// TIA Portal V18 export
// export: Created 2026-06-13T06:09:36.1107387Z, ExportSetting WithDefaults, DisplayName Totally Integrated Automation Portal, DisplayVersion V18, DisplayName TIA Portal Openness, DisplayVersion V18, DisplayName TIA Portal Version Control Interface, DisplayVersion V18, DisplayName STEP 7 Professional, DisplayVersion V18, DisplayName STEP 7 Safety, DisplayVersion V18, DisplayName WinCC Professional, DisplayVersion V18
FUNCTION "FC_HMI_Mirror_PLC2" : Void   // FC41, LAD
{ S7_Optimized_Access := 'TRUE' }
VERSION : 0.1
// stored: AutoNumber true, IsIECCheckEnabled false, SetENOAutomatically false, UDAEnableTagReadback false
BEGIN

REGION Network 1: Mirror AI_V3240_Nuoc_Bon3
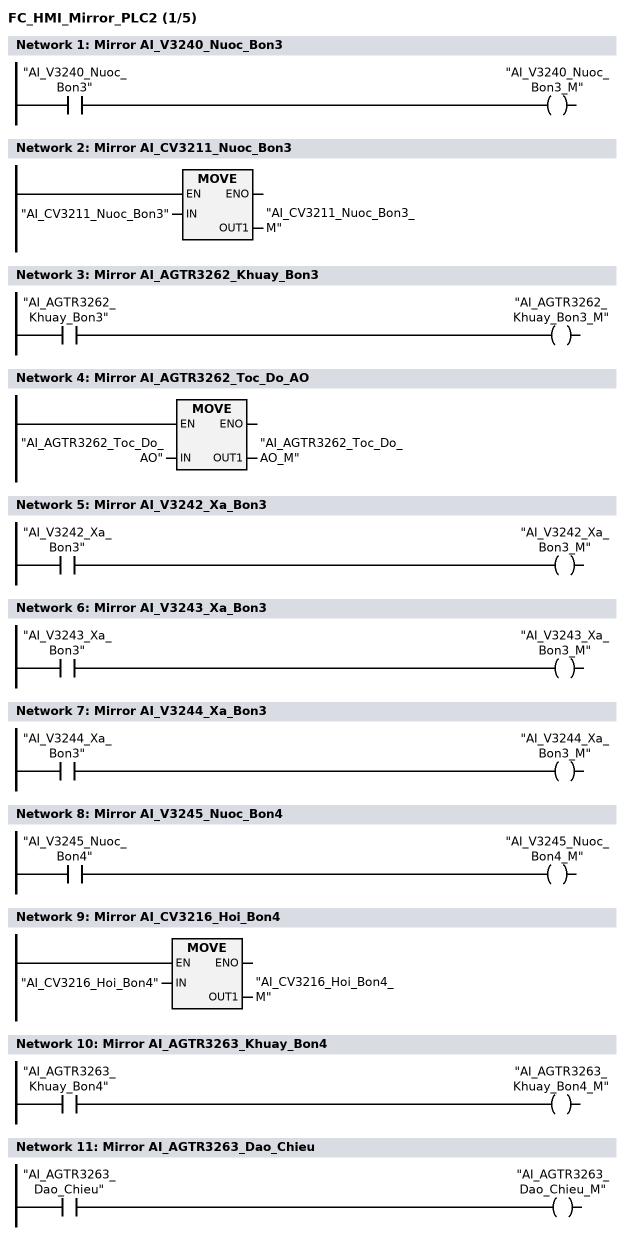
   RUNG wire#powerrail
      Contact( "AI_V3240_Nuoc_Bon3" )
      Coil( "AI_V3240_Nuoc_Bon3_M" )
   END_RUNG
   // the same network as SCL:
   "AI_V3240_Nuoc_Bon3_M" := "AI_V3240_Nuoc_Bon3";
END_REGION

REGION Network 2: Mirror AI_CV3211_Nuoc_Bon3
   RUNG wire#powerrail
      { S7_GenerateENO := "TRUE" } Move(in := "AI_CV3211_Nuoc_Bon3", out1 => "AI_CV3211_Nuoc_Bon3_M")
   END_RUNG
   // the same network as SCL:
   "AI_CV3211_Nuoc_Bon3_M" := "AI_CV3211_Nuoc_Bon3";
END_REGION

REGION Network 3: Mirror AI_AGTR3262_Khuay_Bon3
   RUNG wire#powerrail
      Contact( "AI_AGTR3262_Khuay_Bon3" )
      Coil( "AI_AGTR3262_Khuay_Bon3_M" )
   END_RUNG
   // the same network as SCL:
   "AI_AGTR3262_Khuay_Bon3_M" := "AI_AGTR3262_Khuay_Bon3";
END_REGION

REGION Network 4: Mirror AI_AGTR3262_Toc_Do_AO
   RUNG wire#powerrail
      { S7_GenerateENO := "TRUE" } Move(in := "AI_AGTR3262_Toc_Do_AO", out1 => "AI_AGTR3262_Toc_Do_AO_M")
   END_RUNG
   // the same network as SCL:
   "AI_AGTR3262_Toc_Do_AO_M" := "AI_AGTR3262_Toc_Do_AO";
END_REGION

REGION Network 5: Mirror AI_V3242_Xa_Bon3
   RUNG wire#powerrail
      Contact( "AI_V3242_Xa_Bon3" )
      Coil( "AI_V3242_Xa_Bon3_M" )
   END_RUNG
   // the same network as SCL:
   "AI_V3242_Xa_Bon3_M" := "AI_V3242_Xa_Bon3";
END_REGION

REGION Network 6: Mirror AI_V3243_Xa_Bon3
   RUNG wire#powerrail
      Contact( "AI_V3243_Xa_Bon3" )
      Coil( "AI_V3243_Xa_Bon3_M" )
   END_RUNG
   // the same network as SCL:
   "AI_V3243_Xa_Bon3_M" := "AI_V3243_Xa_Bon3";
END_REGION

REGION Network 7: Mirror AI_V3244_Xa_Bon3
   RUNG wire#powerrail
      Contact( "AI_V3244_Xa_Bon3" )
      Coil( "AI_V3244_Xa_Bon3_M" )
   END_RUNG
   // the same network as SCL:
   "AI_V3244_Xa_Bon3_M" := "AI_V3244_Xa_Bon3";
END_REGION

REGION Network 8: Mirror AI_V3245_Nuoc_Bon4
   RUNG wire#powerrail
      Contact( "AI_V3245_Nuoc_Bon4" )
      Coil( "AI_V3245_Nuoc_Bon4_M" )
   END_RUNG
   // the same network as SCL:
   "AI_V3245_Nuoc_Bon4_M" := "AI_V3245_Nuoc_Bon4";
END_REGION

REGION Network 9: Mirror AI_CV3216_Hoi_Bon4
   RUNG wire#powerrail
      { S7_GenerateENO := "TRUE" } Move(in := "AI_CV3216_Hoi_Bon4", out1 => "AI_CV3216_Hoi_Bon4_M")
   END_RUNG
   // the same network as SCL:
   "AI_CV3216_Hoi_Bon4_M" := "AI_CV3216_Hoi_Bon4";
END_REGION

REGION Network 10: Mirror AI_AGTR3263_Khuay_Bon4
   RUNG wire#powerrail
      Contact( "AI_AGTR3263_Khuay_Bon4" )
      Coil( "AI_AGTR3263_Khuay_Bon4_M" )
   END_RUNG
   // the same network as SCL:
   "AI_AGTR3263_Khuay_Bon4_M" := "AI_AGTR3263_Khuay_Bon4";
END_REGION

REGION Network 11: Mirror AI_AGTR3263_Dao_Chieu
   RUNG wire#powerrail
      Contact( "AI_AGTR3263_Dao_Chieu" )
      Coil( "AI_AGTR3263_Dao_Chieu_M" )
   END_RUNG
   // the same network as SCL:
   "AI_AGTR3263_Dao_Chieu_M" := "AI_AGTR3263_Dao_Chieu";
END_REGION

REGION Network 12: Mirror AI_AGTR3263_Toc_Do_AO
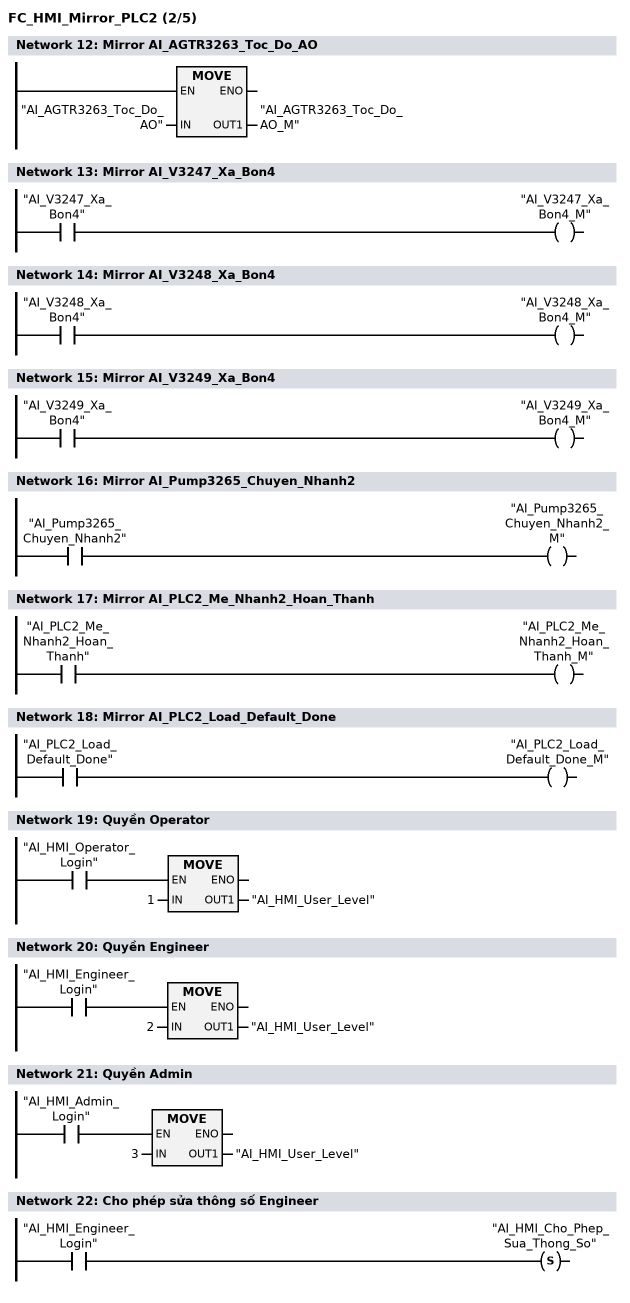
   RUNG wire#powerrail
      { S7_GenerateENO := "TRUE" } Move(in := "AI_AGTR3263_Toc_Do_AO", out1 => "AI_AGTR3263_Toc_Do_AO_M")
   END_RUNG
   // the same network as SCL:
   "AI_AGTR3263_Toc_Do_AO_M" := "AI_AGTR3263_Toc_Do_AO";
END_REGION

REGION Network 13: Mirror AI_V3247_Xa_Bon4
   RUNG wire#powerrail
      Contact( "AI_V3247_Xa_Bon4" )
      Coil( "AI_V3247_Xa_Bon4_M" )
   END_RUNG
   // the same network as SCL:
   "AI_V3247_Xa_Bon4_M" := "AI_V3247_Xa_Bon4";
END_REGION

REGION Network 14: Mirror AI_V3248_Xa_Bon4
   RUNG wire#powerrail
      Contact( "AI_V3248_Xa_Bon4" )
      Coil( "AI_V3248_Xa_Bon4_M" )
   END_RUNG
   // the same network as SCL:
   "AI_V3248_Xa_Bon4_M" := "AI_V3248_Xa_Bon4";
END_REGION

REGION Network 15: Mirror AI_V3249_Xa_Bon4
   RUNG wire#powerrail
      Contact( "AI_V3249_Xa_Bon4" )
      Coil( "AI_V3249_Xa_Bon4_M" )
   END_RUNG
   // the same network as SCL:
   "AI_V3249_Xa_Bon4_M" := "AI_V3249_Xa_Bon4";
END_REGION

REGION Network 16: Mirror AI_Pump3265_Chuyen_Nhanh2
   RUNG wire#powerrail
      Contact( "AI_Pump3265_Chuyen_Nhanh2" )
      Coil( "AI_Pump3265_Chuyen_Nhanh2_M" )
   END_RUNG
   // the same network as SCL:
   "AI_Pump3265_Chuyen_Nhanh2_M" := "AI_Pump3265_Chuyen_Nhanh2";
END_REGION

REGION Network 17: Mirror AI_PLC2_Me_Nhanh2_Hoan_Thanh
   RUNG wire#powerrail
      Contact( "AI_PLC2_Me_Nhanh2_Hoan_Thanh" )
      Coil( "AI_PLC2_Me_Nhanh2_Hoan_Thanh_M" )
   END_RUNG
   // the same network as SCL:
   "AI_PLC2_Me_Nhanh2_Hoan_Thanh_M" := "AI_PLC2_Me_Nhanh2_Hoan_Thanh";
END_REGION

REGION Network 18: Mirror AI_PLC2_Load_Default_Done
   RUNG wire#powerrail
      Contact( "AI_PLC2_Load_Default_Done" )
      Coil( "AI_PLC2_Load_Default_Done_M" )
   END_RUNG
   // the same network as SCL:
   "AI_PLC2_Load_Default_Done_M" := "AI_PLC2_Load_Default_Done";
END_REGION

REGION Network 19: Quyền Operator
   RUNG wire#powerrail
      Contact( "AI_HMI_Operator_Login" )
      { S7_GenerateENO := "TRUE" } Move(in := 1, out1 => "AI_HMI_User_Level")
   END_RUNG
   // the same network as SCL:
   IF "AI_HMI_Operator_Login" THEN "AI_HMI_User_Level" := 1; END_IF;
END_REGION

REGION Network 20: Quyền Engineer
   RUNG wire#powerrail
      Contact( "AI_HMI_Engineer_Login" )
      { S7_GenerateENO := "TRUE" } Move(in := 2, out1 => "AI_HMI_User_Level")
   END_RUNG
   // the same network as SCL:
   IF "AI_HMI_Engineer_Login" THEN "AI_HMI_User_Level" := 2; END_IF;
END_REGION

REGION Network 21: Quyền Admin
   RUNG wire#powerrail
      Contact( "AI_HMI_Admin_Login" )
      { S7_GenerateENO := "TRUE" } Move(in := 3, out1 => "AI_HMI_User_Level")
   END_RUNG
   // the same network as SCL:
   IF "AI_HMI_Admin_Login" THEN "AI_HMI_User_Level" := 3; END_IF;
END_REGION

REGION Network 22: Cho phép sửa thông số Engineer
   RUNG wire#powerrail
      Contact( "AI_HMI_Engineer_Login" )
      S_Coil( "AI_HMI_Cho_Phep_Sua_Thong_So" )
   END_RUNG
   // the same network as SCL:
   IF "AI_HMI_Engineer_Login" THEN "AI_HMI_Cho_Phep_Sua_Thong_So" := TRUE; END_IF;
END_REGION

REGION Network 23: Cho phép sửa thông số Admin
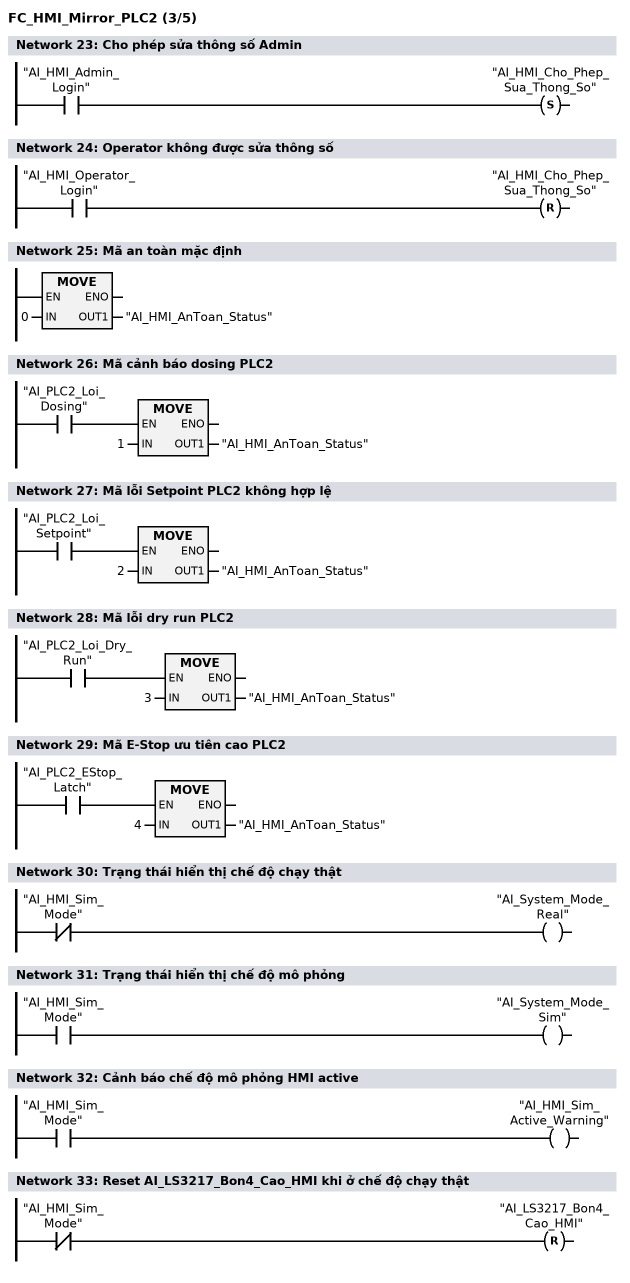
   RUNG wire#powerrail
      Contact( "AI_HMI_Admin_Login" )
      S_Coil( "AI_HMI_Cho_Phep_Sua_Thong_So" )
   END_RUNG
   // the same network as SCL:
   IF "AI_HMI_Admin_Login" THEN "AI_HMI_Cho_Phep_Sua_Thong_So" := TRUE; END_IF;
END_REGION

REGION Network 24: Operator không được sửa thông số
   RUNG wire#powerrail
      Contact( "AI_HMI_Operator_Login" )
      R_Coil( "AI_HMI_Cho_Phep_Sua_Thong_So" )
   END_RUNG
   // the same network as SCL:
   IF "AI_HMI_Operator_Login" THEN "AI_HMI_Cho_Phep_Sua_Thong_So" := FALSE; END_IF;
END_REGION

REGION Network 25: Mã an toàn mặc định
   RUNG wire#powerrail
      { S7_GenerateENO := "TRUE" } Move(in := 0, out1 => "AI_HMI_AnToan_Status")
   END_RUNG
   // the same network as SCL:
   "AI_HMI_AnToan_Status" := 0;
END_REGION

REGION Network 26: Mã cảnh báo dosing PLC2
   RUNG wire#powerrail
      Contact( "AI_PLC2_Loi_Dosing" )
      { S7_GenerateENO := "TRUE" } Move(in := 1, out1 => "AI_HMI_AnToan_Status")
   END_RUNG
   // the same network as SCL:
   IF "AI_PLC2_Loi_Dosing" THEN "AI_HMI_AnToan_Status" := 1; END_IF;
END_REGION

REGION Network 27: Mã lỗi Setpoint PLC2 không hợp lệ
   RUNG wire#powerrail
      Contact( "AI_PLC2_Loi_Setpoint" )
      { S7_GenerateENO := "TRUE" } Move(in := 2, out1 => "AI_HMI_AnToan_Status")
   END_RUNG
   // the same network as SCL:
   IF "AI_PLC2_Loi_Setpoint" THEN "AI_HMI_AnToan_Status" := 2; END_IF;
END_REGION

REGION Network 28: Mã lỗi dry run PLC2
   RUNG wire#powerrail
      Contact( "AI_PLC2_Loi_Dry_Run" )
      { S7_GenerateENO := "TRUE" } Move(in := 3, out1 => "AI_HMI_AnToan_Status")
   END_RUNG
   // the same network as SCL:
   IF "AI_PLC2_Loi_Dry_Run" THEN "AI_HMI_AnToan_Status" := 3; END_IF;
END_REGION

REGION Network 29: Mã E-Stop ưu tiên cao PLC2
   RUNG wire#powerrail
      Contact( "AI_PLC2_EStop_Latch" )
      { S7_GenerateENO := "TRUE" } Move(in := 4, out1 => "AI_HMI_AnToan_Status")
   END_RUNG
   // the same network as SCL:
   IF "AI_PLC2_EStop_Latch" THEN "AI_HMI_AnToan_Status" := 4; END_IF;
END_REGION

REGION Network 30: Trạng thái hiển thị chế độ chạy thật
   RUNG wire#powerrail
      I_Contact( "AI_HMI_Sim_Mode" )
      Coil( "AI_System_Mode_Real" )
   END_RUNG
   // the same network as SCL:
   "AI_System_Mode_Real" := NOT "AI_HMI_Sim_Mode";
END_REGION

REGION Network 31: Trạng thái hiển thị chế độ mô phỏng
   RUNG wire#powerrail
      Contact( "AI_HMI_Sim_Mode" )
      Coil( "AI_System_Mode_Sim" )
   END_RUNG
   // the same network as SCL:
   "AI_System_Mode_Sim" := "AI_HMI_Sim_Mode";
END_REGION

REGION Network 32: Cảnh báo chế độ mô phỏng HMI active
   RUNG wire#powerrail
      Contact( "AI_HMI_Sim_Mode" )
      Coil( "AI_HMI_Sim_Active_Warning" )
   END_RUNG
   // the same network as SCL:
   "AI_HMI_Sim_Active_Warning" := "AI_HMI_Sim_Mode";
END_REGION

REGION Network 33: Reset AI_LS3217_Bon4_Cao_HMI khi ở chế độ chạy thật
   RUNG wire#powerrail
      I_Contact( "AI_HMI_Sim_Mode" )
      R_Coil( "AI_LS3217_Bon4_Cao_HMI" )
   END_RUNG
   // the same network as SCL:
   IF NOT "AI_HMI_Sim_Mode" THEN "AI_LS3217_Bon4_Cao_HMI" := FALSE; END_IF;
END_REGION

REGION Network 34: Reset AI_Pump3265_Chuyen_Nhanh2_Cmd_Nhan_HMI khi ở chế độ chạy thật
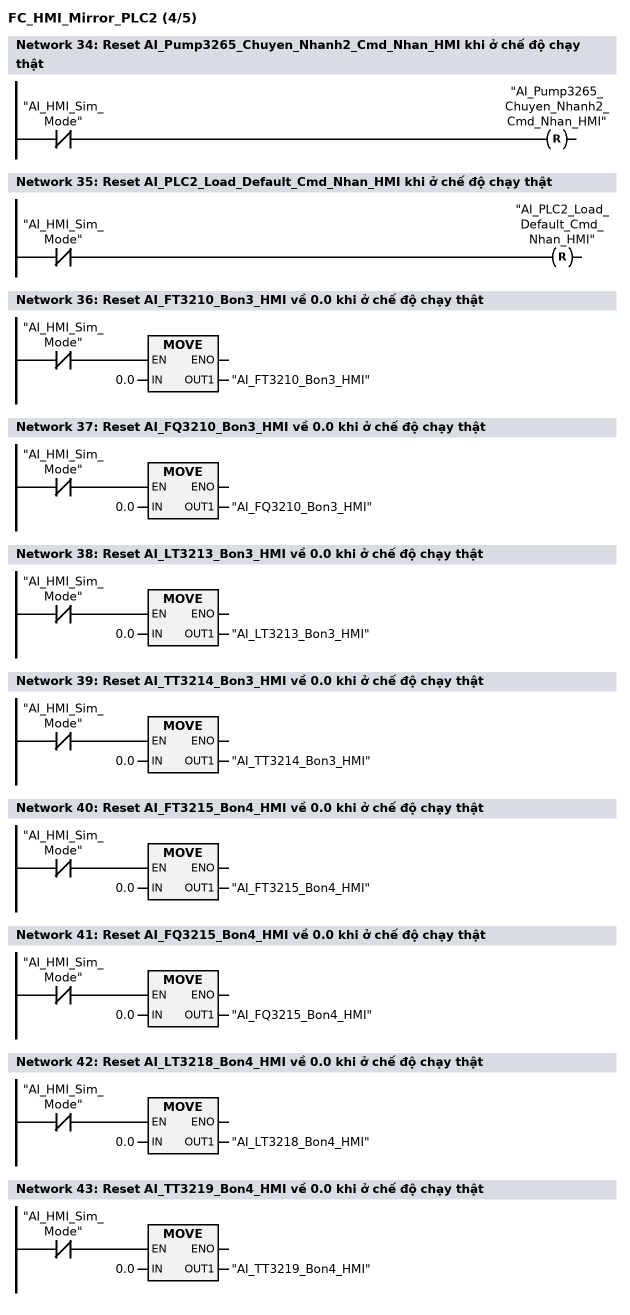
   RUNG wire#powerrail
      I_Contact( "AI_HMI_Sim_Mode" )
      R_Coil( "AI_Pump3265_Chuyen_Nhanh2_Cmd_Nhan_HMI" )
   END_RUNG
   // the same network as SCL:
   IF NOT "AI_HMI_Sim_Mode" THEN "AI_Pump3265_Chuyen_Nhanh2_Cmd_Nhan_HMI" := FALSE; END_IF;
END_REGION

REGION Network 35: Reset AI_PLC2_Load_Default_Cmd_Nhan_HMI khi ở chế độ chạy thật
   RUNG wire#powerrail
      I_Contact( "AI_HMI_Sim_Mode" )
      R_Coil( "AI_PLC2_Load_Default_Cmd_Nhan_HMI" )
   END_RUNG
   // the same network as SCL:
   IF NOT "AI_HMI_Sim_Mode" THEN "AI_PLC2_Load_Default_Cmd_Nhan_HMI" := FALSE; END_IF;
END_REGION

REGION Network 36: Reset AI_FT3210_Bon3_HMI về 0.0 khi ở chế độ chạy thật
   RUNG wire#powerrail
      I_Contact( "AI_HMI_Sim_Mode" )
      { S7_GenerateENO := "TRUE" } Move(in := 0.0, out1 => "AI_FT3210_Bon3_HMI")
   END_RUNG
   // the same network as SCL:
   IF NOT "AI_HMI_Sim_Mode" THEN "AI_FT3210_Bon3_HMI" := 0.0; END_IF;
END_REGION

REGION Network 37: Reset AI_FQ3210_Bon3_HMI về 0.0 khi ở chế độ chạy thật
   RUNG wire#powerrail
      I_Contact( "AI_HMI_Sim_Mode" )
      { S7_GenerateENO := "TRUE" } Move(in := 0.0, out1 => "AI_FQ3210_Bon3_HMI")
   END_RUNG
   // the same network as SCL:
   IF NOT "AI_HMI_Sim_Mode" THEN "AI_FQ3210_Bon3_HMI" := 0.0; END_IF;
END_REGION

REGION Network 38: Reset AI_LT3213_Bon3_HMI về 0.0 khi ở chế độ chạy thật
   RUNG wire#powerrail
      I_Contact( "AI_HMI_Sim_Mode" )
      { S7_GenerateENO := "TRUE" } Move(in := 0.0, out1 => "AI_LT3213_Bon3_HMI")
   END_RUNG
   // the same network as SCL:
   IF NOT "AI_HMI_Sim_Mode" THEN "AI_LT3213_Bon3_HMI" := 0.0; END_IF;
END_REGION

REGION Network 39: Reset AI_TT3214_Bon3_HMI về 0.0 khi ở chế độ chạy thật
   RUNG wire#powerrail
      I_Contact( "AI_HMI_Sim_Mode" )
      { S7_GenerateENO := "TRUE" } Move(in := 0.0, out1 => "AI_TT3214_Bon3_HMI")
   END_RUNG
   // the same network as SCL:
   IF NOT "AI_HMI_Sim_Mode" THEN "AI_TT3214_Bon3_HMI" := 0.0; END_IF;
END_REGION

REGION Network 40: Reset AI_FT3215_Bon4_HMI về 0.0 khi ở chế độ chạy thật
   RUNG wire#powerrail
      I_Contact( "AI_HMI_Sim_Mode" )
      { S7_GenerateENO := "TRUE" } Move(in := 0.0, out1 => "AI_FT3215_Bon4_HMI")
   END_RUNG
   // the same network as SCL:
   IF NOT "AI_HMI_Sim_Mode" THEN "AI_FT3215_Bon4_HMI" := 0.0; END_IF;
END_REGION

REGION Network 41: Reset AI_FQ3215_Bon4_HMI về 0.0 khi ở chế độ chạy thật
   RUNG wire#powerrail
      I_Contact( "AI_HMI_Sim_Mode" )
      { S7_GenerateENO := "TRUE" } Move(in := 0.0, out1 => "AI_FQ3215_Bon4_HMI")
   END_RUNG
   // the same network as SCL:
   IF NOT "AI_HMI_Sim_Mode" THEN "AI_FQ3215_Bon4_HMI" := 0.0; END_IF;
END_REGION

REGION Network 42: Reset AI_LT3218_Bon4_HMI về 0.0 khi ở chế độ chạy thật
   RUNG wire#powerrail
      I_Contact( "AI_HMI_Sim_Mode" )
      { S7_GenerateENO := "TRUE" } Move(in := 0.0, out1 => "AI_LT3218_Bon4_HMI")
   END_RUNG
   // the same network as SCL:
   IF NOT "AI_HMI_Sim_Mode" THEN "AI_LT3218_Bon4_HMI" := 0.0; END_IF;
END_REGION

REGION Network 43: Reset AI_TT3219_Bon4_HMI về 0.0 khi ở chế độ chạy thật
   RUNG wire#powerrail
      I_Contact( "AI_HMI_Sim_Mode" )
      { S7_GenerateENO := "TRUE" } Move(in := 0.0, out1 => "AI_TT3219_Bon4_HMI")
   END_RUNG
   // the same network as SCL:
   IF NOT "AI_HMI_Sim_Mode" THEN "AI_TT3219_Bon4_HMI" := 0.0; END_IF;
END_REGION

REGION Network 44: Mô phỏng truyền thông Modbus TCP: Link Cmd nạp recipe PLC1 sang PLC2_HMI
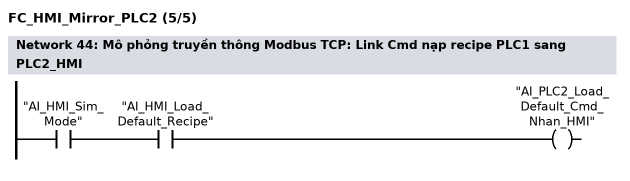
   RUNG wire#powerrail
      Contact( "AI_HMI_Sim_Mode" )
      Contact( "AI_HMI_Load_Default_Recipe" )
      Coil( "AI_PLC2_Load_Default_Cmd_Nhan_HMI" )
   END_RUNG
   // the same network as SCL:
   "AI_PLC2_Load_Default_Cmd_Nhan_HMI" := "AI_HMI_Sim_Mode" AND "AI_HMI_Load_Default_Recipe";
END_REGION
END_FUNCTION
